{attribute addProperty BoxType "KL8519"}
{attribute addProperty Id "StateAT %I*USINT000Data_In_1AT %I*BYTE000Data_In_2AT %I*BYTE000CtrlAT %Q*USINT000LED_Out_green_1AT %Q*BYTE000LED_Out_green_2AT %Q*BYTE000LED_Out_red_1AT %Q*BYTE000LED_Out_red_2AT %Q*BYTE000"}
{attribute addProperty CRC "1223174146"}
{attribute addProperty SizeInBites "0"}
{attribute addProperty SizeInBytes "0"}
TYPE Channel_48E82802 :
STRUCT
	{attribute addProperty Name "State"}
	State AT %I* : USINT;
	{attribute addProperty Name "Data_In_1"}
	Data_In_1 AT %I* : BYTE;
	{attribute addProperty Name "Data_In_2"}
	Data_In_2 AT %I* : BYTE;
	{attribute addProperty Name "Ctrl"}
	Ctrl AT %Q* : USINT;
	{attribute addProperty Name "LED_Out_green_1"}
	LED_Out_green_1 AT %Q* : BYTE;
	{attribute addProperty Name "LED_Out_green_2"}
	LED_Out_green_2 AT %Q* : BYTE;
	{attribute addProperty Name "LED_Out_red_1"}
	LED_Out_red_1 AT %Q* : BYTE;
	{attribute addProperty Name "LED_Out_red_2"}
	LED_Out_red_2 AT %Q* : BYTE;
END_STRUCT
END_TYPE

(* stored: Version 1.2.0.0, ProductVersion 3.1.4024.9
   DUT Channel_48E82802: Id {326f677d-afd5-4130-a039-4c63adf9a777} *)
